// Provides acces to control the light tower components.
FUNCTION_BLOCK FB_LightTower IMPLEMENTS I_LightTower
VAR	
	_redLightControl	: FB_LightTowerComponent;
	_orangeLightControl	: FB_LightTowerComponent;
	_greenLightControl	: FB_LightTowerComponent;
	_buzzerControl		: FB_LightTowerComponent;
END_VAR

// Provides access to buzzer control
PROPERTY Buzzer : I_LightTowerComponent
GET
Buzzer := _buzzerControl;
END_GET
END_PROPERTY

METHOD FB_init : BOOL
VAR_INPUT
	bInitRetains 	: BOOL; // if TRUE, the retain variables are initialized (warm start / cold start)
	bInCopyCode 	: BOOL;  // if TRUE, the instance afterwards gets moved into the copy code (online change)
	greenLight		: REFERENCE TO BOOL;
	orangeLight		: REFERENCE TO BOOL;
	redLight		: REFERENCE TO BOOL;
	buzzer			: REFERENCE TO BOOL;
END_VAR
_greenLightControl.component REF= greenLight;
_orangeLightControl.component REF= orangeLight;
_redLightControl.component REF= redLight;
_buzzerControl.component REF= buzzer;
END_METHOD

// Provides access to green light control
PROPERTY GreenLight : I_LightTowerComponent
GET
GreenLight := _greenLightControl;
END_GET
END_PROPERTY

// Provides access to orange light control
PROPERTY OrangeLight : I_LightTowerComponent
GET
OrangeLight := _orangeLightControl;
END_GET
END_PROPERTY

// Provides access to red light control
PROPERTY RedLight : I_LightTowerComponent
GET
RedLight := _redLightControl;
END_GET
END_PROPERTY

END_FUNCTION_BLOCK

(* stored: Version 1.1.0.1, ProductVersion 3.1.4024.14
   POU FB_LightTower: Id {2aa5c0fe-288c-021a-344a-5de69043f865}, SpecialFunc None
   Property Buzzer: Id {e33b7cba-2bc8-0643-1307-5a8e790efeb7}
   Get Get: Id {edd7e434-922b-0df7-39cf-b632861ed427}
   Method FB_init: Id {c858ca70-8eb9-05d6-173f-4f292f018c10}
   Property GreenLight: Id {b161a0d5-bd03-048e-065b-667b4d9b4d62}
   Get Get: Id {c4ab8bb9-d90e-0b24-0ae2-e6069310aea1}
   Property OrangeLight: Id {cd4856d1-6573-03a9-3545-bf7e18ec6b50}
   Get Get: Id {865508a8-68cf-0f4f-37ff-53b5491578fa}
   Property RedLight: Id {6e098946-9465-0e06-1c58-4ad20da546be}
   Get Get: Id {bbd7d391-ef85-0fa2-273d-a83b936b6c8d} *)
